TYPE EcSoeWrite_Status_typ :
	STRUCT
		bBusy           : BOOL;
        bError          : BOOL;
	END_STRUCT
END_TYPE

(* stored: Version 1.1.0.1, ProductVersion 3.1.4024.3
   DUT EcSoeWrite_Status_typ: Id {36767477-7714-0348-0130-c2576fedfa72} *)
